// TIA Portal V18 export
TYPE "RCS_SysComInterface_V1"
// stored: IsFailsafeCompliant false
   STRUCT
      CPUFristCycle : Bool;   // CPU start frist cycle
      SysRun : Bool;   // Safety OK & Control On
      Reset : Bool;   // Station total Reset signial
      EstopOK : Bool;   // Station total Estop signial
      SafetyDoorOK : Bool;   // Station all Safety door status OK
      LightCurtainOK : Bool;   // Station all light curtain status OK
      SetInitial : Bool;   // Station total initial signal
      InitialRun : Bool;   // Station total initial running signal
      Ready : Bool;   // Station in AutoMode and all Status OK, ready for AutoRuning
      ManualMode : Bool;   // Station in Manual Mode
      Auto : "RCS_SysAuto_V1";
   END_STRUCT;
END_TYPE
